TEXTLIST textListTop
  0 = ''
  1 = 'X'
  2 = 'V '
  3 = 'Λ'
   = ''
END_TEXTLIST

(* stored: Version 1.1.0.1, ProductVersion 3.1.4024.11
   TextList textListTop: Id {876c4917-c231-0cdf-0caa-adfbedff56c8} *)
